FUNCTION fIntExtFun : real
VAR_INPUT
	Range:ARRAY[1..2] OF REAL;
	resolution:DINT;//number of integration rectangles
END_VAR
VAR
	i:DINT;
	Xi,MDi:REAL;
	IntegrationStep: REAL;
END_VAR

IF Resolution<>0 THEN
	//calcular el paso de integracion
	IntegrationStep:=(Range[2]-Range[1])/DINT_TO_REAL(Resolution);
	
	FOR i := 1 TO resolution DO
		Xi := DINT_TO_REAL(i)*IntegrationStep;//paso de integracion actual
		MDi :=Extfun(Xi) ;//llamada a la funcion abstracta
		fIntegrateMf := fIntExtFun + MDi*IntegrationStep;
	END_FOR
END_IF

END_FUNCTION

(* stored: Version 1.1.0.1, ProductVersion 3.1.4024.6
   POU fIntExtFun: Id {e41cdefd-9837-43f8-9489-7da9063df70c}, SpecialFunc None *)
